FUNCTION VolNow : REAL

VolNow := GVL.tank_area * GVL.high_now;

END_FUNCTION

(* stored: Version 1.1.0.1, ProductVersion 3.1.4024.12
   POU VolNow: Id {77c24618-b925-4840-a558-accae81d177a}, SpecialFunc None *)
